// TIA Portal V20 export
VAR_GLOBAL   // PLC tag table "11_Settings"
END_VAR
VAR_GLOBAL CONSTANT   // user constants
   MAX_NO_OF_DEVICES_IRT : Int := 200;
   MAX_NO_OF_MODULES_IRT : Int := 200;
   MAX_NO_OF_DEVICES_RT : Int := 200;
   MAX_NO_OF_MODULES_RT : Int := 200;
END_VAR
